// TIA Portal V18 export
FUNCTION_BLOCK "DelayDirChange"   // FB61, FBD
{ S7_Optimized_Access := 'TRUE' }
VERSION : 0.1
// stored: AutoNumber true, IsIECCheckEnabled false, IsRetainMemResEnabled false, MemoryReserve 100, SetENOAutomatically false, UDAEnableTagReadback false
   VAR_INPUT
      pt : Time := T#2S;
      dirFwd : Bool;
      dirRev : Bool;
   END_VAR
   VAR_OUTPUT
      qFwd : Bool;
      qRev : Bool;
      block : Bool;
   END_VAR
   VAR
      tonfwd { S7_SetPoint := 'True'} : TON_TIME;
      tonrev { S7_SetPoint := 'True'} : TON_TIME;
      block_fwd : Bool;
   END_VAR
   VAR_TEMP
      wait_done : Bool;
      block_rev : Bool;
   END_VAR
BEGIN

REGION Network 2
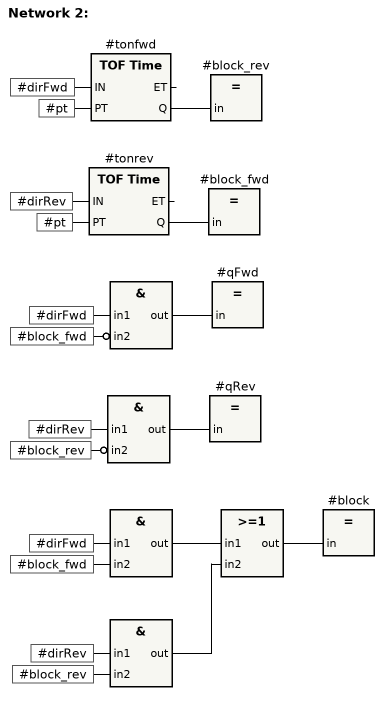
   #tonfwd(IN := #dirFwd, PT := #pt);   // TOF
   #block_rev := #tonfwd.Q;
   #tonrev(IN := #dirRev, PT := #pt);   // TOF
   #block_fwd := #tonrev.Q;
   #qFwd := #dirFwd AND NOT #block_fwd;
   #qRev := #dirRev AND NOT #block_rev;
   #block := (#dirFwd AND #block_fwd) OR (#dirRev AND #block_rev);
END_REGION
END_FUNCTION_BLOCK
